FUNCTION_BLOCK FB_NOTT_ICS
VAR_INPUT
END_VAR
VAR_OUTPUT
END_VAR
VAR
	
	Delay_Lines:		FB_NOTT_DELAY_LINES;
	
	Shutters:			FB_NOTT_SHUTTERS;
	
	TipTilt:			FB_NOTT_TipTilt;
	

	
	
END_VAR



Delay_Lines();
Delay_Lines.M_SET_DL_ACTUAL_POS();

Shutters();

TipTilt();

END_FUNCTION_BLOCK

(* stored: Version 1.1.0.1, ProductVersion 3.1.4024.12
   POU FB_NOTT_ICS: Id {35e04548-ee92-4622-970e-d83afc0b7c18}, SpecialFunc None *)
